// Library/POUs/Additional/MC_ActivateNextCommand/Structures/ActivateNextCommandRecvData
{attribute 'pack_mode' := '1'} 
// ------------------------------------------------------------------------- 
//  SRCI Robot Library                                                
// ------------------------------------------------------------------------- 
//                                                                           
//  Object:      ActivateNextCommandRecvData                                       
//  Author:      Thorsten Brach                                                
//  Date:        2024-06-01
//
//  Description:                                              
//   
//                                                                           
//  Copyright: 
//    (C) 2024 Thorsten Brach. All rights reserved                                                                                                                                            
//             Licensed under the LGPL-3.0 license.
//                                                                           
//  Disclaimer:                                                                           
//    This project is provided without any guarantee and can be used for   
//    private and commercial purposes. Any use is at the user’s 
//    own risk and responsibility.
//
// -------------------------------------------------------------------------
TYPE ActivateNextCommandRecvData EXTENDS RspHeader :
STRUCT
  /// Relates to ListenerID >0
  /// Number of successful trigger -based command invocations
  /// For more information refer to chapter 5.5.12.4.
  InvocationCounter  : USINT;
  /// Reserve
  Reserve            : SINT;
  /// Unique system-generated ID of the "Action" when the function is triggered.
  /// • >0: The "Action" is started by the trigger function with identical FollowID.
  /// • <0: The "Action" is stopped by the trigger function with identical FollowID.
  /// For more information see chapter 5.5.12.4 EmitterID, ListenerID, FollowID and OriginID
  OriginID           : INT;
END_STRUCT
END_TYPE

// Library/POUs/Additional/MC_ActivateNextCommand/Structures/ActivateNextCommandSendData
{attribute 'pack_mode' := '1'}
// ------------------------------------------------------------------------- 
//  SRCI Robot Library                                                
// ------------------------------------------------------------------------- 
//                                                                           
//  Object:      ActivateNextCommandParCmd                                       
//  Author:      Thorsten Brach                                                
//  Date:        2024-06-01
//
//  Description:                                              
//   
//                                                                           
//  Copyright: 
//    (C) 2024 Thorsten Brach. All rights reserved                                                                                                                                            
//             Licensed under the LGPL-3.0 license.
//                                                                           
//  Disclaimer:                                                                           
//    This project is provided without any guarantee and can be used for   
//    private and commercial purposes. Any use is at the user’s 
//    own risk and responsibility.
//
// -------------------------------------------------------------------------
TYPE ActivateNextCommandSendData EXTENDS CmdHeader:   
STRUCT  
  /// ID of Action that will be executed when this command is active
  /// • >0: Start Action        - Start executing the Action function with the identical ListenerID.
  /// • <0: Stop Action         - Stop executing the Action function with the identical ListenerID.
  /// •  0: Undefined (default) - If no EmitterID is defined, the function returns an error message
  /// For more information see chapter 5.5.12.4
  EmitterID  : ARRAY[0..3] OF SINT;  
  /// ID of the trigger function that may be triggered:
  /// • 0: Immediately (default). - Start executing THIS function immediately.
  /// • >0: Triggero Start executing when the trigger function with the identical EmitterID is called.
  /// For more information see chapter 5.5.12.4.
  ListenerID : SINT;
  /// Reserve
  Reserve    : BYTE;
END_STRUCT
END_TYPE

// Library/POUs/Additional/MC_AvoidSingularity/Structures/AvoidSingularityOutCmd
{attribute 'pack_mode' := '1'} 
// ------------------------------------------------------------------------- 
//  SRCI Robot Library                                                
// ------------------------------------------------------------------------- 
//                                                                           
//  Object:      AvoidSingularityOutCmd                                       
//  Author:      Thorsten Brach                                                
//  Date:        2024-06-22
//
//  Description:                                              
//   
//                                                                           
//  Copyright: 
//    (C) 2024 Thorsten Brach. All rights reserved                                                                                                                                            
//             Licensed under the LGPL-3.0 license.
//                                                                           
//  Disclaimer:                                                                           
//    This project is provided without any guarantee and can be used for   
//    private and commercial purposes. Any use is at the user’s 
//    own risk and responsibility.
//
// -------------------------------------------------------------------------
TYPE AvoidSingularityOutCmd :
STRUCT
END_STRUCT
END_TYPE

// Library/POUs/Additional/MC_AvoidSingularity/Structures/AvoidSingularityParCmd
{attribute 'pack_mode' := '1'} 
// ------------------------------------------------------------------------- 
//  SRCI Robot Library                                                
// ------------------------------------------------------------------------- 
//                                                                           
//  Object:      AvoidSingularityParCmd                                       
//  Author:      Thorsten Brach                                                
//  Date:        2024-06-22
//
//  Description:                                              
//   
//                                                                           
//  Copyright: 
//    (C) 2024 Thorsten Brach. All rights reserved                                                                                                                                            
//             Licensed under the LGPL-3.0 license.
//                                                                           
//  Disclaimer:                                                                           
//    This project is provided without any guarantee and can be used for   
//    private and commercial purposes. Any use is at the user’s 
//    own risk and responsibility.
//
// -------------------------------------------------------------------------
TYPE AvoidSingularityParCmd :
STRUCT
  /// Define in which way the singularity should be avoided
  Mode : SingularityAvoidanceMode; 
END_STRUCT
END_TYPE

// Library/POUs/Additional/MC_AvoidSingularity/Structures/AvoidSingularityRecvData
{attribute 'pack_mode' := '1'} 
// ------------------------------------------------------------------------- 
//  SRCI Robot Library                                                
// ------------------------------------------------------------------------- 
//                                                                           
//  Object:      AvoidSingularityRecvData                                       
//  Author:      Thorsten Brach                                                
//  Date:        2024-06-22
//
//  Description:                                              
//   
//                                                                           
//  Copyright: 
//    (C) 2024 Thorsten Brach. All rights reserved                                                                                                                                            
//             Licensed under the LGPL-3.0 license.
//                                                                           
//  Disclaimer:                                                                           
//    This project is provided without any guarantee and can be used for   
//    private and commercial purposes. Any use is at the user’s 
//    own risk and responsibility.
//
// -------------------------------------------------------------------------
TYPE AvoidSingularityRecvData EXTENDS RspHeader :
STRUCT
  /// TRUE when robot is set to RA power state "Enabled".
  Enabled : BOOL;
END_STRUCT
END_TYPE

// Library/POUs/Additional/MC_AvoidSingularity/Structures/AvoidSingularitySendData
{attribute 'pack_mode' := '1'}
// ------------------------------------------------------------------------- 
//  SRCI Robot Library                                                
// ------------------------------------------------------------------------- 
//                                                                           
//  Object:      AvoidSingularitySendData                                       
//  Author:      Thorsten Brach                                                
//  Date:        2024-06-22
//
//  Description:                                              
//   
//                                                                           
//  Copyright: 
//    (C) 2024 Thorsten Brach. All rights reserved                                                                                                                                            
//             Licensed under the LGPL-3.0 license.
//                                                                           
//  Disclaimer:                                                                           
//    This project is provided without any guarantee and can be used for   
//    private and commercial purposes. Any use is at the user’s 
//    own risk and responsibility.
//
// -------------------------------------------------------------------------
TYPE AvoidSingularitySendData EXTENDS CmdHeader: 
STRUCT
  /// Set TRUE to activate avoid singularity mode
  Enable : BOOL;
  /// Define in which way the singularity should be avoided
  Mode   : SingularityAvoidanceMode;
END_STRUCT
END_TYPE

// Library/POUs/Additional/MC_BrakeTest/Structures/BrakeTestOutCmd
{attribute 'pack_mode' := '1'} 
// ------------------------------------------------------------------------- 
//  SRCI Robot Library                                                
// ------------------------------------------------------------------------- 
//                                                                           
//  Object:      BrakeTestOutCmd                                       
//  Author:      Thorsten Brach                                                
//  Date:        2024-06-01
//
//  Description:                                              
//   
//                                                                           
//  Copyright: 
//    (C) 2024 Thorsten Brach. All rights reserved                                                                                                                                            
//             Licensed under the LGPL-3.0 license.
//                                                                           
//  Disclaimer:                                                                           
//    This project is provided without any guarantee and can be used for   
//    private and commercial purposes. Any use is at the user’s 
//    own risk and responsibility.
//
// -------------------------------------------------------------------------
TYPE BrakeTestOutCmd :
STRUCT
  /// Indicates the result of the brake test of the robot axes related to the brake test.
  /// • TRUE: The brake test has been realized successfully.
  /// • FALSE: The brake test failed. 
  /// See Table 6-735 for bit assignment.
  RobotAxesStatus    : RobotAxesFlags;
  /// Indicates the result of the brake test of the external robot axes related to the brake test.
  /// • TRUE: The brake test has been realized successfully.
  /// • FALSE: The brake test failed.
  /// See Table 6-735 for bit assignment.
  ExternalAxesStatus : ExternalAxesFlags;
  /// Indicates the warning messages availability related to the brake functionality of the robot axes reported by the RC.
  /// • TRUE: One or more warning messages are available.
  /// • FALSE: No warning message is available.
  /// See Table 6-735 for bit assignment.
  RobotAxesWarning   : RobotAxesFlags;
  /// Indicates the warning messages availability related to the brake functionality of the external robot axis reported by the RC.
  /// • TRUE: One or more warning messages are available.
  /// • FALSE: No warning message is available.
  /// See Table 6-735 for bit assignment.
  ExternalAxesWarning: ExternalAxesFlags;
END_STRUCT
END_TYPE

// Library/POUs/Additional/MC_BrakeTest/Structures/BrakeTestParCmd
{attribute 'pack_mode' := '1'} 
// ------------------------------------------------------------------------- 
//  SRCI Robot Library                                                
// ------------------------------------------------------------------------- 
//                                                                           
//  Object:      BrakeTestParCmd                                       
//  Author:      Thorsten Brach                                                
//  Date:        2024-06-01
//
//  Description:                                              
//   
//                                                                           
//  Copyright: 
//    (C) 2024 Thorsten Brach. All rights reserved                                                                                                                                            
//             Licensed under the LGPL-3.0 license.
//                                                                           
//  Disclaimer:                                                                           
//    This project is provided without any guarantee and can be used for   
//    private and commercial purposes. Any use is at the user’s 
//    own risk and responsibility.
//
// -------------------------------------------------------------------------
TYPE BrakeTestParCmd :
STRUCT
  /// Parameter which determines the behavior towards the previously sent and still active or buffered commands.
  AbortingMode       : AbortingMode;
  /// Defines which of the robot axis should be activated for the brake test.
  /// • TRUE (default): Axis activated.
  /// • FALSE: Axis deactivated.
  /// See Table 6-735 for bit assignment.
  RobotAxesActive    : RobotAxesFlags;
  /// Defines which of the external robot axis should be activated for the brake test.
  /// • TRUE: Axis activated.
  /// • FALSE (default): Axis deactivated.
  /// See Table 6-735 for bit assignment.   
  ExternalAxesActive : ExternalAxesFlags;
  /// Defines the target sequence in which the command will be executed
  SequenceFlag       : SequenceFlag;
END_STRUCT
END_TYPE

// Library/POUs/Additional/MC_BrakeTest/Structures/BrakeTestRecvData
{attribute 'pack_mode' := '1'} 
// ------------------------------------------------------------------------- 
//  SRCI Robot Library                                                
// ------------------------------------------------------------------------- 
//                                                                           
//  Object:      BrakeTestRecvData                                       
//  Author:      Thorsten Brach                                                
//  Date:        2024-06-01
//
//  Description:                                              
//   
//                                                                           
//  Copyright: 
//    (C) 2024 Thorsten Brach. All rights reserved                                                                                                                                            
//             Licensed under the LGPL-3.0 license.
//                                                                           
//  Disclaimer:                                                                           
//    This project is provided without any guarantee and can be used for   
//    private and commercial purposes. Any use is at the user’s 
//    own risk and responsibility.
//
// -------------------------------------------------------------------------
TYPE BrakeTestRecvData EXTENDS RspHeader :
STRUCT
  /// Indicates the result of the brake test of the robot axes related to the brake test.
  /// • TRUE: The brake test has been realized successfully.
  /// • FALSE: The brake test failed. 
  /// See Table 6-735 for bit assignment.
  RobotAxesStatus    : BYTE;
  /// Indicates the result of the brake test of the external robot axes related to the brake test.
  /// • TRUE: The brake test has been realized successfully.
  /// • FALSE: The brake test failed.
  /// See Table 6-735 for bit assignment.
  ExternalAxesStatus : BYTE;
  /// Indicates the warning messages availability related to the brake functionality of the robot axes reported by the RC.
  /// • TRUE: One or more warning messages are available.
  /// • FALSE: No warning message is available.
  /// See Table 6-735 for bit assignment.
  RobotAxesWarning   : BYTE;
  /// Indicates the warning messages availability related to the brake functionality of the external robot axis reported by the RC.
  /// • TRUE: One or more warning messages are available.
  /// • FALSE: No warning message is available.
  /// See Table 6-735 for bit assignment.
  ExternalAxesWarning: BYTE;
END_STRUCT
END_TYPE

// Library/POUs/Additional/MC_BrakeTest/Structures/BrakeTestSendData
{attribute 'pack_mode' := '1'}
// ------------------------------------------------------------------------- 
//  SRCI Robot Library                                                
// ------------------------------------------------------------------------- 
//                                                                           
//  Object:      BrakeTestSendData                                       
//  Author:      Thorsten Brach                                                
//  Date:        2024-06-01
//
//  Description:                                              
//   
//                                                                           
//  Copyright: 
//    (C) 2024 Thorsten Brach. All rights reserved                                                                                                                                            
//             Licensed under the LGPL-3.0 license.
//                                                                           
//  Disclaimer:                                                                           
//    This project is provided without any guarantee and can be used for   
//    private and commercial purposes. Any use is at the user’s 
//    own risk and responsibility.
//
// -------------------------------------------------------------------------
TYPE BrakeTestSendData EXTENDS CmdHeader:   
STRUCT
  /// Defines which of the robot axis should be activated for the brake test.
  /// • TRUE (default): Axis activated.
  /// • FALSE: Axis deactivated.
  /// See Table 6-735 for bit assignment.
  RobotAxesActive    : BYTE;
  /// Defines which of the external robot axis should be activated for the brake test.
  /// • TRUE: Axis activated.
  /// • FALSE (default): Axis deactivated.
  /// See Table 6-735 for bit assignment.   
  ExternalAxesActive : BYTE; 
END_STRUCT
END_TYPE

// Library/POUs/Additional/MC_CallSubprogram/Structures/CallSubprogramOutCmd
{attribute 'pack_mode' := '1'} 
// ------------------------------------------------------------------------- 
//  SRCI Robot Library                                                
// ------------------------------------------------------------------------- 
//                                                                           
//  Object:      CallSubprogramOutCmd                                       
//  Author:      Thorsten Brach                                                
//  Date:        2024-08-03
//
//  Description:                                              
//   
//                                                                           
//  Copyright: 
//    (C) 2024 Thorsten Brach. All rights reserved                                                                                                                                            
//             Licensed under the LGPL-3.0 license.
//                                                                           
//  Disclaimer:                                                                           
//    This project is provided without any guarantee and can be used for   
//    private and commercial purposes. Any use is at the user’s 
//    own risk and responsibility.
//
// -------------------------------------------------------------------------
TYPE CallSubprogramOutCmd :
STRUCT
  /// Unique, system-generated ID of the instance of CallSubprogram. 
  /// Can be used to specifically stop instance of a subprogram via the function Stop Subprogram (chapter 6.5.21) 
  /// if multiinstancing  is supported by RC 
  InstanceID         : DINT; 
  /// Unique system-generated ID of the "Action" when the function is triggered.
  /// • >0: The "Action" is started by the trigger function with identical FollowID.
  /// • <0: The "Action" is stopped by the trigger function with identical FollowID.
  /// For more information see chapter 5.5.12.4 EmitterID, ListenerID, FollowID and OriginID
  OriginID           : INT;
  /// Relates to ListenerID >0
  /// Number of successful trigger -based command invocations
  /// For more information refer to chapter 5.5.12.4.
  InvocationCounter  : USINT;
  /// The requested subprogram on the RC is in progress. Movement of the axes trough this subprogram is possible.
  InProgress         : BOOL;
  /// Acyclic output parameters of the subprogram Array length adjusts to transmitted data (max 190 bytes)
  ReturnData         : ARRAY[0..RobotLibraryParameter.SUB_PROGRAM_DATA_MAX] OF BYTE;
END_STRUCT
END_TYPE

// Library/POUs/Additional/MC_CallSubprogram/Structures/CallSubprogramParCmd
{attribute 'pack_mode' := '1'} 
// ------------------------------------------------------------------------- 
//  SRCI Robot Library                                                
// ------------------------------------------------------------------------- 
//                                                                           
//  Object:      CallSubprogramParCmd                                       
//  Author:      Thorsten Brach                                                
//  Date:        2024-08-03
//
//  Description:                                              
//   
//                                                                           
//  Copyright: 
//    (C) 2024 Thorsten Brach. All rights reserved                                                                                                                                            
//             Licensed under the LGPL-3.0 license.
//                                                                           
//  Disclaimer:                                                                           
//    This project is provided without any guarantee and can be used for   
//    private and commercial purposes. Any use is at the user’s 
//    own risk and responsibility.
//
// -------------------------------------------------------------------------
TYPE CallSubprogramParCmd :
STRUCT
  /// Program number of the subprogram in the RC
  JobID             : UINT;
  /// ID of associated trigger function:
  /// • 0: No Trigger (default) - No trigger related behavior
  /// • >0: Triggero - Start executing when the trigger function with the identical EmitterID is triggered.
  /// Always positive.
  /// For more information, see chapter 5.5.12 Triggers
  ListenerID        : SINT;
  /// Acyclic input parameters of the subprogram Array length adjusts to transmitted data (max 190 bytes)
  Data              : ARRAY[0..RobotLibraryParameter.SUB_PROGRAM_DATA_MAX] OF BYTE;
END_STRUCT
END_TYPE

// Library/POUs/Additional/MC_CallSubprogram/Structures/CallSubprogramRecvData
{attribute 'pack_mode' := '1'} 
// ------------------------------------------------------------------------- 
//  SRCI Robot Library                                                
// ------------------------------------------------------------------------- 
//                                                                           
//  Object:      CallSubprogramRecvData                                       
//  Author:      Thorsten Brach                                                
//  Date:        2024-08-03
//
//  Description:                                              
//   
//                                                                           
//  Copyright: 
//    (C) 2024 Thorsten Brach. All rights reserved                                                                                                                                            
//             Licensed under the LGPL-3.0 license.
//                                                                           
//  Disclaimer:                                                                           
//    This project is provided without any guarantee and can be used for   
//    private and commercial purposes. Any use is at the user’s 
//    own risk and responsibility.
//
// -------------------------------------------------------------------------
TYPE CallSubprogramRecvData EXTENDS RspHeader :
STRUCT
  /// Relates to ListenerID >0
  /// Number of successful trigger-based command invocations - For more information refer TO chapter 5.5.12.4
  InvocationCounter : USINT;  
  /// Reserve
  Reserve           : SINT;
  /// Unique system-generated ID of the "Action" when the function is triggered.
  /// • >0: The "Action" is started by the trigger funcrion with identical FollowID.
  /// • <0: The "Action" is stopped by the trigger function with identical FollowID.
  /// For more information see chapter 5.5.12.4 EmitterID, ListenerID, FollowID and OriginID
  OriginID          : INT;
  /// Percentage of already traversed distance of current job.
  /// If not supported : • -1
  Progress          : UINT;
  /// The requested subprogram on the RC is in progress. Movement of the axes trough this subprogram is possible.
  InProgress        : BOOL;
  /// Acyclic output parameters of the subprogram Array length adjusts to transmitted data (max 190 bytes)
  ReturnData        : ARRAY[0..RobotLibraryParameter.SUB_PROGRAM_DATA_MAX] OF BYTE;  
END_STRUCT
END_TYPE

// Library/POUs/Additional/MC_CallSubprogram/Structures/CallSubprogramSendData
{attribute 'pack_mode' := '1'}
// ------------------------------------------------------------------------- 
//  SRCI Robot Library                                                
// ------------------------------------------------------------------------- 
//                                                                           
//  Object:      CallSubprogramSendData                                       
//  Author:      Thorsten Brach                                                
//  Date:        2024-08-03
//
//  Description:                                              
//   
//                                                                           
//  Copyright: 
//    (C) 2024 Thorsten Brach. All rights reserved                                                                                                                                            
//             Licensed under the LGPL-3.0 license.
//                                                                           
//  Disclaimer:                                                                           
//    This project is provided without any guarantee and can be used for   
//    private and commercial purposes. Any use is at the user’s 
//    own risk and responsibility.
//
// -------------------------------------------------------------------------
TYPE CallSubprogramSendData EXTENDS CmdHeader: 
STRUCT
  /// ID of Action that will be executed when this command is active
  /// • >0: Start Action - Start executing the Action function with the identical ListenerID.
  /// • <0: Stop Action  -  Stop executing the Action function with the identical ListenerID.
  /// • 0: No trigger (default)-  If no EmitterID is defined, the function will not trigger any Action during its execution
  /// For more information see section Triggers of this chapter or chapter 5.5.12.4.
  EmitterID          : ARRAY [0..3] OF SINT;  
  /// ID of associated trigger function:
  /// • 0: No Trigger (default) - No trigger related behavior
  /// • >0: Triggero - Start executing when the trigger function with the identical EmitterID is triggered.
  /// Always positive.
  /// For more information, see chapter 5.5.12 Triggers
  ListenerID        : SINT;
  /// Reserve
  Reserve           : BYTE;
  /// Program number of the subprogram in the RC
  JobID             : UINT;
  /// Acyclic input parameters of the subprogram Array length adjusts to transmitted data (max 190 bytes)
  Data              : ARRAY[0..RobotLibraryParameter.SUB_PROGRAM_DATA_MAX] OF BYTE;
END_STRUCT
END_TYPE

// Library/POUs/Additional/MC_CollisionDetection/Structures/CollisionDetectionOutCmd
{attribute 'pack_mode' := '1'} 
// ------------------------------------------------------------------------- 
//  SRCI Robot Library                                                
// ------------------------------------------------------------------------- 
//                                                                           
//  Object:      CollisionDetectionOutCmd                                       
//  Author:      Thorsten Brach                                                
//  Date:        2024-06-22
//
//  Description:                                              
//   
//                                                                           
//  Copyright: 
//    (C) 2024 Thorsten Brach. All rights reserved                                                                                                                                            
//             Licensed under the LGPL-3.0 license.
//                                                                           
//  Disclaimer:                                                                           
//    This project is provided without any guarantee and can be used for   
//    private and commercial purposes. Any use is at the user’s 
//    own risk and responsibility.
//
// -------------------------------------------------------------------------
TYPE CollisionDetectionOutCmd :
STRUCT
END_STRUCT
END_TYPE

// Library/POUs/Additional/MC_CollisionDetection/Structures/CollisionDetectionParCmd
{attribute 'pack_mode' := '1'} 
// ------------------------------------------------------------------------- 
//  SRCI Robot Library                                                
// ------------------------------------------------------------------------- 
//                                                                           
//  Object:      CollisionDetectionParCmd                                       
//  Author:      Thorsten Brach                                                
//  Date:        2024-06-22
//
//  Description:                                              
//   
//                                                                           
//  Copyright: 
//    (C) 2024 Thorsten Brach. All rights reserved                                                                                                                                            
//             Licensed under the LGPL-3.0 license.
//                                                                           
//  Disclaimer:                                                                           
//    This project is provided without any guarantee and can be used for   
//    private and commercial purposes. Any use is at the user’s 
//    own risk and responsibility.
//
// -------------------------------------------------------------------------
TYPE CollisionDetectionParCmd :
STRUCT
  /// Processing mode
  ProcessingMode     : ProcessingMode;
  ///  Defines the robot behavior after detecting the collision (at least one option must be supported):
  ReactionMode       : CollisionReactionMode;
  /// Set TRUE to activate and FALSE to deactivate "CollisionDetection".
  /// Default: TRUE
  ActivateMonitoring : BOOL;
  /// Defines the type of threshold setting (at least one option must be supported)
  ThresholdMode      : ThresholdMode;
  /// Defines the level of sensitivity of all axes.
  /// • 0..99: Sensitivity lower than robot vendor default. 
  ///          At minimum value "0" there is no sensitivity. The lower the value, the lower the sensitivity at the collision detection.
  /// • 100 (default): The value is aligned with the robot vendor-specific default value.
  /// • 101..200: Sensitivity higher than robot vendor default. At maximum value "200" highest possible sensitivity at the collision detection.
  Sensitivity        : REAL;
  /// Defines the level of sensitivity of the respective axis.
  /// Values:
  /// • 0..99: Sensitivity lower than robot vendor default. At minimum value "0" there is no sensitivity and collision detection for the respective axis. 
  ///          The lower the value, the lower the sensitivity at the collision detection.
  /// • 100 (default): The value is aligned with the robot vendor-specific default value.
  /// • 101..200: Sensitivity higher than robot vendor default. At maximum value "200" highest possible sensitivity at the collision detection.
  /// Index:
  /// • [0]: J1 First joint of the robot.
  /// • [1]: J2 Second joint of the robot.
  /// • [2] J3 Third joint of the robot.
  /// • [3] J4 Forth joint of the robot.
  /// • [4] J5 Fifth joint of the robot.
  /// • [5] J6 Six joint of the robot.
  /// • [6] J7 Seventh joint of the robot, if willbe used.
  SensitivityAxis    : ARRAY[0..6] OF REAL;
  /// Relates to "ThresholdMode" Manual. Defines the threshold of the torque for each robot axis. If the threshold is exceeded, the RA stops.
  /// Index:
  /// • [0] J1 First joint of the robot.
  /// • [1] J2 Second joint of the robot.
  /// • [2] J3 Third joint of the robot.
  /// • [3] J4 Forth joint of the robot.
  /// • [4] J5 Fifth joint of the robot.
  /// • [5] J6 Six joint of the robot.
  /// • [6] J7 Seventh joint of the robot, if will be used
  LimitAxis          : ARRAY[0..6] OF REAL;
  /// Relates to "LimitAxis". Defines the unit of the threshold.
  /// • [0]: Percentage (%) (default) O
  /// • [1]: Newton meter (Nm). O
  /// • [2] Milliampere (mA).
  UnitLimitAxis      : USINT;
  /// Defines the target sequence in which the command will be executed
  SequenceFlag       : SequenceFlag;
END_STRUCT
END_TYPE

// Library/POUs/Additional/MC_CollisionDetection/Structures/CollisionDetectionRecvData
{attribute 'pack_mode' := '1'} 
// ------------------------------------------------------------------------- 
//  SRCI Robot Library                                                
// ------------------------------------------------------------------------- 
//                                                                           
//  Object:      CollisionDetectionRecvData                                       
//  Author:      Thorsten Brach                                                
//  Date:        2024-06-22
//
//  Description:                                              
//   
//                                                                           
//  Copyright: 
//    (C) 2024 Thorsten Brach. All rights reserved                                                                                                                                            
//             Licensed under the LGPL-3.0 license.
//                                                                           
//  Disclaimer:                                                                           
//    This project is provided without any guarantee and can be used for   
//    private and commercial purposes. Any use is at the user’s 
//    own risk and responsibility.
//
// -------------------------------------------------------------------------
TYPE CollisionDetectionRecvData EXTENDS RspHeader :
STRUCT
END_STRUCT
END_TYPE

// Library/POUs/Additional/MC_CollisionDetection/Structures/CollisionDetectionSendData
{attribute 'pack_mode' := '1'}
// ------------------------------------------------------------------------- 
//  SRCI Robot Library                                                
// ------------------------------------------------------------------------- 
//                                                                           
//  Object:      CollisionDetectionSendData                                       
//  Author:      Thorsten Brach                                                
//  Date:        2024-06-22
//
//  Description:                                              
//   
//                                                                           
//  Copyright: 
//    (C) 2024 Thorsten Brach. All rights reserved                                                                                                                                            
//             Licensed under the LGPL-3.0 license.
//                                                                           
//  Disclaimer:                                                                           
//    This project is provided without any guarantee and can be used for   
//    private and commercial purposes. Any use is at the user’s 
//    own risk and responsibility.
//
// -------------------------------------------------------------------------
TYPE CollisionDetectionSendData EXTENDS CmdHeader: 
STRUCT
  /// Set TRUE to activate and FALSE to deactivate "CollisionDetection".
  /// Default: TRUE
  ActivateMonitoring : BOOL;
  /// Relates to "LimitAxis". Defines the unit of the threshold.
  /// • [0]: Percentage (%) (default) O
  /// • [1]: Newton meter (Nm). O
  /// • [2] Milliampere (mA).
  UnitLimitAxis      : USINT;
  /// Defines the type of threshold setting (at least one option must be supported)
  ThresholdMode      : ThresholdMode;
  ///  Defines the robot behavior after detecting the collision (at least one option must be supported):
  ReactionMode       : CollisionReactionMode;
  /// Defines the level of sensitivity of all axes.
  /// • 0..99: Sensitivity lower than robot vendor default. 
  ///          At minimum value "0" there is no sensitivity. The lower the value, the lower the sensitivity at the collision detection.
  /// • 100 (default): The value is aligned with the robot vendor-specific default value.
  /// • 101..200: Sensitivity higher than robot vendor default. At maximum value "200" highest possible sensitivity at the collision detection.
  Sensitivity        : INT;
  /// Defines the level of sensitivity of the respective axis.
  /// Values:
  /// • 0..99: Sensitivity lower than robot vendor default. At minimum value "0" there is no sensitivity and collision detection for the respective axis. 
  ///          The lower the value, the lower the sensitivity at the collision detection.
  /// • 100 (default): The value is aligned with the robot vendor-specific default value.
  /// • 101..200: Sensitivity higher than robot vendor default. At maximum value "200" highest possible sensitivity at the collision detection.
  /// Index:
  /// • [0]: J1 First joint of the robot.
  /// • [1]: J2 Second joint of the robot.
  /// • [2] J3 Third joint of the robot.
  /// • [3] J4 Forth joint of the robot.
  /// • [4] J5 Fifth joint of the robot.
  /// • [5] J6 Six joint of the robot.
  /// • [6] J7 Seventh joint of the robot, if willbe used.
  SensitivityAxis    : ARRAY[0..6] OF INT;

  /// Relates to "ThresholdMode" Manual. Defines the threshold of the torque for each robot axis. If the threshold is exceeded, the RA stops.
  /// Index:
  /// • [0] J1 First joint of the robot.
  /// • [1] J2 Second joint of the robot.
  /// • [2] J3 Third joint of the robot.
  /// • [3] J4 Forth joint of the robot.
  /// • [4] J5 Fifth joint of the robot.
  /// • [5] J6 Six joint of the robot.
  /// • [6] J7 Seventh joint of the robot, if will be used
  LimitAxis          : ARRAY[0..6] OF REAL;
END_STRUCT
END_TYPE

// Library/POUs/Additional/MC_ExchangeConfiguration/Structures/ExchangeConfigurationOutCmd
{attribute 'pack_mode' := '1'} 
// ------------------------------------------------------------------------- 
//  SRCI Robot Library                                                
// ------------------------------------------------------------------------- 
//                                                                           
//  Object:      ExchangeConfigurationOutCmd                                       
//  Author:      Thorsten Brach                                                
//  Date:        2024-06-22
//
//  Description:                                              
//   
//                                                                           
//  Copyright: 
//    (C) 2024 Thorsten Brach. All rights reserved                                                                                                                                            
//             Licensed under the LGPL-3.0 license.
//                                                                           
//  Disclaimer:                                                                           
//    This project is provided without any guarantee and can be used for   
//    private and commercial purposes. Any use is at the user’s 
//    own risk and responsibility.
//
// -------------------------------------------------------------------------
TYPE ExchangeConfigurationOutCmd :
STRUCT
  /// Returns a metric of how many CMDs it can receive and manage at the same time
  LengthACR                 : UINT;
  /// Highest index of available tools on the RC.
  HighestToolIndex          : USINT;
  /// Highest index of available frames on the RC.
  HighestFrameIndex         : USINT;
  /// Highest index of available loads on the RC.
  HighestLoadIndex          : USINT;
  /// Highest index of available work areas on the RC.
  HighestWorkAreaIndex      : USINT;
  /// Datas which are synchronized
  DataInSync                : DataInSync;
  /// Index of tool changed on RC
  ChangeIndexTool           : USINT;
  /// Index of frame changed on RC
  ChangeIndexFrame          : USINT;
  /// Index of load changed on RC
  ChangeIndexLoad           : USINT;
  ///Index of work area changed on RC
  ChangeIndexWorkArea       : USINT;
  /// Working hours of an RA connected to the RC
  RAWorkingHours            : UDINT;
  /// Signals that a brake test is required in the defined monitoring time (see chapter 6.5.27)
  BrakeTestRequired         : BOOL;
  /// StepMode is active and set to ExactStop (see chapter 6.1.3)
  StepModeExactStopActive   : BOOL;
  /// StepMode is active and set to Blending (see chapter 6.1.3)
  StepModeBlendingActive    : BOOL;
  /// PathAccuracyMode is active (see chapter 6.5.22)
  PathAccuracyMode          : BOOL;
  /// AvoidSingularity is active (see chapter 6.5.23)
  AvoidSingularity          : BOOL;
  /// CollisionDetection is active (see chapter 6.5.35)
  CollisionDetectionEnabled : BOOL;
  /// Cyclic dynamics status bit Accelerating is supported by RC (see chapter 5.5.3.2)
  AcceleratingSupported     : BOOL;
  /// Cyclic dynamics status bit Decelerating is supported by RC (see chapter 5.5.3.2)
  DecceleratingSupported    : BOOL;
  /// Cyclic dynamics status bit ConstantVelocity is supported by RC (see chapter 5.5.3.2)
  ConstantVelocitySupported : BOOL;
  /// Total system hours of an RA connected to the RC. Must not be modifiable by the user.
  /// •  0: Invalid
  /// • >1: Total system hours
  RCWorkingHours            : UDINT;
END_STRUCT
END_TYPE

// Library/POUs/Additional/MC_ExchangeConfiguration/Structures/ExchangeConfigurationParCmd
{attribute 'pack_mode' := '1'} 
// ------------------------------------------------------------------------- 
//  SRCI Robot Library                                                
// ------------------------------------------------------------------------- 
//                                                                           
//  Object:      ExchangeConfigurationParCmd                                       
//  Author:      Thorsten Brach                                                
//  Date:        2024-06-22
//
//  Description:                                              
//   
//                                                                           
//  Copyright: 
//    (C) 2024 Thorsten Brach. All rights reserved                                                                                                                                            
//             Licensed under the LGPL-3.0 license.
//                                                                           
//  Disclaimer:                                                                           
//    This project is provided without any guarantee and can be used for   
//    private and commercial purposes. Any use is at the user’s 
//    own risk and responsibility.
//
// -------------------------------------------------------------------------
TYPE ExchangeConfigurationParCmd :
STRUCT
  /// Defines up to which level of severity messages will be logged in the RC's server log
  LogLevel                   : LogLevel;
  /// Defines blending behavior for single move commands. One of the optional modes must be supported.
  ///  • 0 (default): Move to end position
  ///       Robot moves exactly the target position independently of the selected "BlendingMode"
  ///  • 1: Wait at blending parameter 
  ///       Robot stops its movement when the specified blending parameter is reached
  WaitAtBlendingZone         : BOOL;
  /// Allow a sequence switch from primary to secondary while a subprogram called via CallSubprogram (6.5.18) in the sequence is in progress
  AllowSecSeqWhileSubprogram : BOOL;
  /// Allows blending when CallSubprogram is called in sequence and removed afterwards. For more information see chapter 6.5.21.
  /// • 0 (default): Dynamic blending is prevented
  /// • 1: Dynamic blending is allowed
  AllowDynamicBlending       : BOOL;
  /// Defines waiting time of RC between receiving a first move command when motion queue is empty and starting the first movement. See also chapter 5.6.8.
  DelayTime                  : UINT;
  /// Define number of points required to calculate the blending. See also chapter 5.6.8.
  WaitForNrOfCmd             : UINT;
  /// Maximum allowed time between incrementation of LifeSign before communication error.
  /// • <10 ms: Invalid
  /// • 50 ms: default
  /// See also chapter 5.6.6.2.
  LifeSignTimeOut            : UINT;
  /// Defines a delay time between detecting an inconsistency of configuration data between server and client and executing the defined SyncReaction. 
  /// Always positive. Default: 0 ms
  SyncDelay                  : UINT;
  /// Specifies system reaction in case inconsistency of synchronization data is detected according to Table 6-81. For more information refer to chapter 5.6.7.2
  SyncReaction               : SyncReaction;
  /// Datas which are synchronized
  DataInSync                 : DataInSync;
  /// Enable datas to synchronize
  DataEnableSync             : DataEnableSync;
END_STRUCT
END_TYPE

// Library/POUs/Additional/MC_ExchangeConfiguration/Structures/ExchangeConfigurationRecvData
{attribute 'pack_mode' := '1'} 
// ------------------------------------------------------------------------- 
//  SRCI Robot Library                                                
// ------------------------------------------------------------------------- 
//                                                                           
//  Object:      ExchangeConfigurationRecvData                                       
//  Author:      Thorsten Brach                                                
//  Date:        2024-06-22
//
//  Description:                                              
//   
//                                                                           
//  Copyright: 
//    (C) 2024 Thorsten Brach. All rights reserved                                                                                                                                            
//             Licensed under the LGPL-3.0 license.
//                                                                           
//  Disclaimer:                                                                           
//    This project is provided without any guarantee and can be used for   
//    private and commercial purposes. Any use is at the user’s 
//    own risk and responsibility.
//
// -------------------------------------------------------------------------
TYPE ExchangeConfigurationRecvData EXTENDS RspHeader :
STRUCT
  /// TRUE when function is exchanging data
  Enabled                   : BOOL;
  /// Reserve 
  Reserve1                  : BYTE;
   /// Returns a metric of how many CMDs it can receive and manage at the same time
  LengthACR                 : UINT;
  /// Highest index of available tools on the RC.
  HighestToolIndex          : USINT;
  /// Highest index of available frames on the RC.
  HighestFrameIndex         : USINT;
  /// Highest index of available loads on the RC.
  HighestLoadIndex          : USINT;
  /// Highest index of available work areas on the RC.
  HighestWorkAreaIndex      : USINT; 
  /// Datas which are synchronized
  DataInSync                : DataInSync;
  /// Reserve 
  Reserve2                  : BYTE;
  /// Index of tool changed on RC
  ChangeIndexTool           : USINT;
  /// Index of frame changed on RC
  ChangeIndexFrame          : USINT;
  /// Index of load changed on RC
  ChangeIndexLoad           : USINT;
  ///Index of work area changed on RC
  ChangeIndexWorkArea       : USINT;
  /// Working hours of an RA connected to the RC
  RAWorkingHours            : UDINT;
  /// Status byte
  StatusByte                : BYTE;
  /// Cyclic dynamics status bit ConstantVelocity is supported by RC (see chapter 5.5.3.2)
  ConstantVelocitySupported : BOOL;
  /// Total system hours of an RA connected to the RC. Must not be modifiable by the user.
  /// •  0: Invalid
  /// • >1: Total system hours
  RCWorkingHours            : UDINT;
END_STRUCT
END_TYPE

// Library/POUs/Additional/MC_ExchangeConfiguration/Structures/ExchangeConfigurationSendData
{attribute 'pack_mode' := '1'}
// ------------------------------------------------------------------------- 
//  SRCI Robot Library                                                
// ------------------------------------------------------------------------- 
//                                                                           
//  Object:      ExchangeConfigurationSendData                                       
//  Author:      Thorsten Brach                                                
//  Date:        2024-06-22
//
//  Description:                                              
//   
//                                                                           
//  Copyright: 
//    (C) 2024 Thorsten Brach. All rights reserved                                                                                                                                            
//             Licensed under the LGPL-3.0 license.
//                                                                           
//  Disclaimer:                                                                           
//    This project is provided without any guarantee and can be used for   
//    private and commercial purposes. Any use is at the user’s 
//    own risk and responsibility.
//
// -------------------------------------------------------------------------
TYPE ExchangeConfigurationSendData EXTENDS CmdHeader: 
STRUCT
  /// Defines up to which level of severity messages will be logged in the RC's server log
  LogLevel                   : LogLevel;
  /// Miscellaneous control bits 
  CtrlByte                   : BYTE;
  /// Defines waiting time of RC between receiving a first move command when motion queue is empty and starting the first movement. See also chapter 5.6.8.
  DelayTime                  : UINT;
  /// Define number of points required to calculate the blending. See also chapter 5.6.8.
  WaitForNrOfCmd             : UINT;
  /// Maximum allowed time between incrementation of LifeSign before communication error.
  /// • <10 ms: Invalid
  /// • 50 ms: default
  /// See also chapter 5.6.6.2.
  LifeSignTimeOut            : UINT;
  /// Defines a delay time between detecting an inconsistency of configuration data between server and client and executing the defined SyncReaction. 
  /// Always positive. Default: 0 ms
  SyncDelay                  : UINT;
  /// Specifies system reaction in case inconsistency of synchronization data is detected according to Table 6-81. For more information refer to chapter 5.6.7.2
  SyncReaction               : SyncReaction;
  /// Datas which are synchronized
  DataInSync                 : DataInSync;
  /// Reserve
  Reserve1                   : BYTE;
  /// Enable datas to synchronize
  DataEnableSync             : DataEnableSync;  
  /// Reserve
  Reserve2                   : BYTE;
END_STRUCT
END_TYPE

// Library/POUs/Additional/MC_FreeDrive/Structures/FreeDriveOutCmd
{attribute 'pack_mode' := '1'} 
// ------------------------------------------------------------------------- 
//  SRCI Robot Library                                                
// ------------------------------------------------------------------------- 
//                                                                           
//  Object:      FreeDriveOutCmd                                       
//  Author:      Thorsten Brach                                                
//  Date:        2024-06-22
//
//  Description:                                              
//   
//                                                                           
//  Copyright: 
//    (C) 2024 Thorsten Brach. All rights reserved                                                                                                                                            
//             Licensed under the LGPL-3.0 license.
//                                                                           
//  Disclaimer:                                                                           
//    This project is provided without any guarantee and can be used for   
//    private and commercial purposes. Any use is at the user’s 
//    own risk and responsibility.
//
// -------------------------------------------------------------------------
TYPE FreeDriveOutCmd :
STRUCT
  /// TRUE when function is exchanging data
  Enabled                   : BOOL;
  /// Returns a metric of how many CMDs it can receive and manage at the same time
  LengthACR                 : UINT;
  /// Highest index of available tools on the RC.
  HighestToolIndex          : USINT;
  /// Highest index of available frames on the RC.
  HighestFrameIndex         : USINT;
  /// Highest index of available loads on the RC.
  HighestLoadIndex          : USINT;
  /// Highest index of available work areas on the RC.
  HighestWorkAreaIndex      : USINT;
  /// Datas which are synchronized
  DataInSync                : DataInSync;
  /// Index of tool changed on RC
  ChangeIndexTool           : USINT;
  /// Index of frame changed on RC
  ChangeIndexFrame          : USINT;
  /// Index of load changed on RC
  ChangeIndexLoad           : USINT;
  ///Index of work area changed on RC
  ChangeIndexWorkArea       : USINT;
  /// Working hours of an RA connected to the RC
  RAWorkingHours            : UDINT;
  /// Signals that a brake test is required in the defined monitoring time (see chapter 6.5.27)
  BrakeTestRequired         : BOOL;
  /// StepMode is active and set to ExactStop (see chapter 6.1.3)
  StepModeExactStopActive   : BOOL;
  /// StepMode is active and set to Blending (see chapter 6.1.3)
  StepModeBlendingActive    : BOOL;
  /// PathAccuracyMode is active (see chapter 6.5.22)
  PathAccuracyMode          : BOOL;
  /// AvoidSingularity is active (see chapter 6.5.23)
  AvoidSingularity          : BOOL;
  /// CollisionDetection is active (see chapter 6.5.35)
  CollisionDetectionEnabled : BOOL;
  /// Cyclic dynamics status bit Accelerating is supported by RC (see chapter 5.5.3.2)
  AcceleratingSupported     : BOOL;
  /// Cyclic dynamics status bit Decelerating is supported by RC (see chapter 5.5.3.2)
  DecceleratingSupported    : BOOL;
  /// Cyclic dynamics status bit ConstantVelocity is supported by RC (see chapter 5.5.3.2)
  ConstantVelocitySupported : BOOL;
  /// Total system hours of an RA connected to the RC. Must not be modifiable by the user.
  /// •  0: Invalid
  /// • >1: Total system hours
  RCWorkingHours            : UDINT;
END_STRUCT
END_TYPE

// Library/POUs/Additional/MC_FreeDrive/Structures/FreeDriveParCmd
{attribute 'pack_mode' := '1'} 
// ------------------------------------------------------------------------- 
//  SRCI Robot Library                                                
// ------------------------------------------------------------------------- 
//                                                                           
//  Object:      FreeDriveParCmd                                       
//  Author:      Thorsten Brach                                                
//  Date:        2024-06-22
//
//  Description:                                              
//   
//                                                                           
//  Copyright: 
//    (C) 2024 Thorsten Brach. All rights reserved                                                                                                                                            
//             Licensed under the LGPL-3.0 license.
//                                                                           
//  Disclaimer:                                                                           
//    This project is provided without any guarantee and can be used for   
//    private and commercial purposes. Any use is at the user’s 
//    own risk and responsibility.
//
// -------------------------------------------------------------------------
TYPE FreeDriveParCmd :
STRUCT
  /// Defines up to which level of severity messages will be logged in the RC's server log
  LogLevel                   : LogLevel;
  /// Defines blending behavior for single move commands. One of the optional modes must be supported.
  ///  • 0 (default): Move to end position
  ///       Robot moves exactly the target position independently of the selected "BlendingMode"
  ///  • 1: Wait at blending parameter 
  ///       Robot stops its movement when the specified blending parameter is reached
  WaitAtBlendingZone         : BOOL;
  /// Allow a sequence switch from primary to secondary while a subprogram called via CallSubprogram (6.5.18) in the sequence is in progress
  AllowSecSeqWhileSubprogram : BOOL;
  /// ToDo
  AllowDynamicBlending       : BOOL;
  /// Defines waiting time of RC between receiving a first move command when motion queue is empty and starting the first movement. See also chapter 5.6.8.
  DelayTime                  : UINT;
  /// Define number of points required to calculate the blending. See also chapter 5.6.8.
  WaitForNrOfCmd             : UINT;
  /// Maximum allowed time between incrementation of LifeSign before communication error.
  /// • <10 ms: Invalid
  /// • 50 ms: default
  /// See also chapter 5.6.6.2.
  LifeSignTimeOut            : UINT;
  /// Defines a delay time between detecting an inconsistency of configuration data between server and client and executing the defined SyncReaction. 
  /// Always positive. Default: 0 ms
  SyncDelay                  : UINT;
  /// Specifies system reaction in case inconsistency of synchronization data is detected according to Table 6-81. For more information refer to chapter 5.6.7.2
  SyncReaction               : SyncReaction;
  /// Datas which are synchronized
  DataInSync                 : DataInSync;
  /// Enable datas to synchronize
  DataEnableSync             : DataEnableSync;
END_STRUCT
END_TYPE

// Library/POUs/Additional/MC_FreeDrive/Structures/FreeDriveRecvData
{attribute 'pack_mode' := '1'} 
// ------------------------------------------------------------------------- 
//  SRCI Robot Library                                                
// ------------------------------------------------------------------------- 
//                                                                           
//  Object:      FreeDriveRecvData                                       
//  Author:      Thorsten Brach                                                
//  Date:        2024-06-22
//
//  Description:                                              
//   
//                                                                           
//  Copyright: 
//    (C) 2024 Thorsten Brach. All rights reserved                                                                                                                                            
//             Licensed under the LGPL-3.0 license.
//                                                                           
//  Disclaimer:                                                                           
//    This project is provided without any guarantee and can be used for   
//    private and commercial purposes. Any use is at the user’s 
//    own risk and responsibility.
//
// -------------------------------------------------------------------------
TYPE FreeDriveRecvData EXTENDS RspHeader :
STRUCT
  /// TRUE when function is exchanging data
  Enabled                   : BOOL;
END_STRUCT
END_TYPE

// Library/POUs/Additional/MC_FreeDrive/Structures/FreeDriveSendData
{attribute 'pack_mode' := '1'}
// ------------------------------------------------------------------------- 
//  SRCI Robot Library                                                
// ------------------------------------------------------------------------- 
//                                                                           
//  Object:      FreeDriveSendData                                       
//  Author:      Thorsten Brach                                                
//  Date:        2024-06-22
//
//  Description:                                              
//   
//                                                                           
//  Copyright: 
//    (C) 2024 Thorsten Brach. All rights reserved                                                                                                                                            
//             Licensed under the LGPL-3.0 license.
//                                                                           
//  Disclaimer:                                                                           
//    This project is provided without any guarantee and can be used for   
//    private and commercial purposes. Any use is at the user’s 
//    own risk and responsibility.
//
// -------------------------------------------------------------------------
TYPE FreeDriveSendData EXTENDS CmdHeader: 
STRUCT
  /// Set TRUE to activate "FreeDrive".
  Enable            : BOOL;
END_STRUCT
END_TYPE

// Library/POUs/Additional/MC_MeasuringInput/Structures/MeasuringInputOutCmd
{attribute 'pack_mode' := '1'} 
// ------------------------------------------------------------------------- 
//  SRCI Robot Library                                                
// ------------------------------------------------------------------------- 
//                                                                           
//  Object:      MeasuringInputOutCmd                                       
//  Author:      Thorsten Brach                                                
//  Date:        2024-06-21
//
//  Description:                                              
//   
//                                                                           
//  Copyright: 
//    (C) 2024 Thorsten Brach. All rights reserved                                                                                                                                            
//             Licensed under the LGPL-3.0 license.
//                                                                           
//  Disclaimer:                                                                           
//    This project is provided without any guarantee and can be used for   
//    private and commercial purposes. Any use is at the user’s 
//    own risk and responsibility.
//
// -------------------------------------------------------------------------
TYPE MeasuringInputOutCmd :
STRUCT
  /// FB is returning a unique ID for the called measurement.
  MeasuringID        : UINT;
  /// Measured robot position value at the rising edge of the digital input in selected coordinate systems (see input parameters ToolNo and FrameNo).
  Measurings         : ARRAY[1..2] OF MeasuringInputResult;  
END_STRUCT
END_TYPE

// Library/POUs/Additional/MC_MeasuringInput/Structures/MeasuringInputParCmd
{attribute 'pack_mode' := '1'} 
// ------------------------------------------------------------------------- 
//  SRCI Robot Library                                                
// ------------------------------------------------------------------------- 
//                                                                           
//  Object:      MeasuringInputParCmd                                       
//  Author:      Thorsten Brach                                                
//  Date:        2024-06-21
//
//  Description:                                              
//   
//                                                                           
//  Copyright: 
//    (C) 2024 Thorsten Brach. All rights reserved                                                                                                                                            
//             Licensed under the LGPL-3.0 license.
//                                                                           
//  Disclaimer:                                                                           
//    This project is provided without any guarantee and can be used for   
//    private and commercial purposes. Any use is at the user’s 
//    own risk and responsibility.
//
// -------------------------------------------------------------------------
TYPE MeasuringInputParCmd :
STRUCT
  /// Type of measurement (at least one option must be supported):
  MeasuringMode      : MeasuringIoMode;
  /// Specifies the desired digital input register. 
  /// More information about the different periphery register can be found in chapter 6.4
  Index              : USINT;
  ///Specifies the desired bit in the digital input register, that should be read. 
  /// More information about the different periphery register can be found in chapter 6.4.
  BitNumber          : USINT;
END_STRUCT
END_TYPE

// Library/POUs/Additional/MC_MeasuringInput/Structures/MeasuringInputRecvData
{attribute 'pack_mode' := '1'} 
// ------------------------------------------------------------------------- 
//  SRCI Robot Library                                                
// ------------------------------------------------------------------------- 
//                                                                           
//  Object:      MeasuringInputRecvData                                       
//  Author:      Thorsten Brach                                                
//  Date:        2024-06-21
//
//  Description:                                              
//   
//                                                                           
//  Copyright: 
//    (C) 2024 Thorsten Brach. All rights reserved                                                                                                                                            
//             Licensed under the LGPL-3.0 license.
//                                                                           
//  Disclaimer:                                                                           
//    This project is provided without any guarantee and can be used for   
//    private and commercial purposes. Any use is at the user’s 
//    own risk and responsibility.
//
// -------------------------------------------------------------------------
TYPE MeasuringInputRecvData EXTENDS RspHeader :
STRUCT
  /// FB is returning a unique ID for the called measurement.
  MeasuringID        : UINT;
  /// Measured robot position value at the rising edge of the digital input in selected coordinate systems (see input parameters ToolNo and FrameNo).
  Measurings         : ARRAY[1..2] OF MeasuringInputResult;  
END_STRUCT
END_TYPE

// Library/POUs/Additional/MC_MeasuringInput/Structures/MeasuringInputSendData
{attribute 'pack_mode' := '1'}
// ------------------------------------------------------------------------- 
//  SRCI Robot Library                                                
// ------------------------------------------------------------------------- 
//                                                                           
//  Object:      MeasuringInputSendData                                       
//  Author:      Thorsten Brach                                                
//  Date:        2024-06-21
//
//  Description:                                              
//   
//                                                                           
//  Copyright: 
//    (C) 2024 Thorsten Brach. All rights reserved                                                                                                                                            
//             Licensed under the LGPL-3.0 license.
//                                                                           
//  Disclaimer:                                                                           
//    This project is provided without any guarantee and can be used for   
//    private and commercial purposes. Any use is at the user’s 
//    own risk and responsibility.
//
// -------------------------------------------------------------------------
TYPE MeasuringInputSendData EXTENDS CmdHeader:   
STRUCT
  /// Type of measurement (at least one option must be supported):
  MeasuringMode      : MeasuringIoMode;
  /// Specifies the desired digital input register. 
  /// More information about the different periphery register can be found in chapter 6.4
  Index              : USINT;
  ///Specifies the desired bit in the digital input register, that should be read. 
  /// More information about the different periphery register can be found in chapter 6.4.
  BitNumber          : USINT;
END_STRUCT
END_TYPE

// Library/POUs/Additional/MC_OpenBrake/Structures/OpenBrakeOutCmd
{attribute 'pack_mode' := '1'} 
// ------------------------------------------------------------------------- 
//  SRCI Robot Library                                                
// ------------------------------------------------------------------------- 
//                                                                           
//  Object:      BrakeTestOutCmd                                       
//  Author:      Thorsten Brach                                                
//  Date:        2024-06-01
//
//  Description:                                              
//   
//                                                                           
//  Copyright: 
//    (C) 2024 Thorsten Brach. All rights reserved                                                                                                                                            
//             Licensed under the LGPL-3.0 license.
//                                                                           
//  Disclaimer:                                                                           
//    This project is provided without any guarantee and can be used for   
//    private and commercial purposes. Any use is at the user’s 
//    own risk and responsibility.
//
// -------------------------------------------------------------------------
TYPE OpenBrakeOutCmd :
STRUCT
  /// TRUE when "OpenBrake" is active.
  Enabled                   : BOOL;  
  /// Indicates the brake release status of the main robot axes.
  /// • TRUE: The brake of the axis is opened.
  /// • FALSE: The brake of the axis is closed.
  /// See Table 6-735 for bit assignment
  RobotAxesBrakeReleased    : RobotAxesFlags;
  /// Indicates the brake release status of the external robot axes.
  /// • TRUE: The brake of the axis is opened.
  /// • FALSE: The brake of the axis is closed/not supported
  /// See Table 6-735 for bit assignment
  ExternalAxesBrakeReleased : ExternalAxesFlags;
END_STRUCT
END_TYPE

// Library/POUs/Additional/MC_OpenBrake/Structures/OpenBrakeParCmd
{attribute 'pack_mode' := '1'} 
// ------------------------------------------------------------------------- 
//  SRCI Robot Library                                                
// ------------------------------------------------------------------------- 
//                                                                           
//  Object:      OpenBrakeParCmd                                       
//  Author:      Thorsten Brach                                                
//  Date:        2024-06-01
//
//  Description:                                              
//   
//                                                                           
//  Copyright: 
//    (C) 2024 Thorsten Brach. All rights reserved                                                                                                                                            
//             Licensed under the LGPL-3.0 license.
//                                                                           
//  Disclaimer:                                                                           
//    This project is provided without any guarantee and can be used for   
//    private and commercial purposes. Any use is at the user’s 
//    own risk and responsibility.
//
// -------------------------------------------------------------------------
TYPE OpenBrakeParCmd :
STRUCT
  /// Defines which brake of the robot axes must be released.
  /// • TRUE: Open the brake of the axis.
  /// • FALSE (default): Close the brake of the axis.
  RobotAxesBrakeRelease    : RobotAxesFlags;
  /// Defines which brake of the external robot axis must be released.
  /// • TRUE: Open the brake of the axis.
  /// • FALSE (default): Close the brake of the axis.
  /// See Table 6-676 for bit assignment.
  ExternalAxesBrakeRelease : ExternalAxesFlags;
END_STRUCT
END_TYPE

// Library/POUs/Additional/MC_OpenBrake/Structures/OpenBrakeRecvData
{attribute 'pack_mode' := '1'} 
// ------------------------------------------------------------------------- 
//  SRCI Robot Library                                                
// ------------------------------------------------------------------------- 
//                                                                           
//  Object:      BrakeTestRecvData                                       
//  Author:      Thorsten Brach                                                
//  Date:        2024-06-01
//
//  Description:                                              
//   
//                                                                           
//  Copyright: 
//    (C) 2024 Thorsten Brach. All rights reserved                                                                                                                                            
//             Licensed under the LGPL-3.0 license.
//                                                                           
//  Disclaimer:                                                                           
//    This project is provided without any guarantee and can be used for   
//    private and commercial purposes. Any use is at the user’s 
//    own risk and responsibility.
//
// -------------------------------------------------------------------------
TYPE OpenBrakeRecvData EXTENDS RspHeader :
STRUCT
  /// TRUE when "OpenBrake" is active.
  Enabled                   : BYTE;  
  /// Indicates the brake release status of the main robot axes.
  /// • TRUE: The brake of the axis is opened.
  /// • FALSE: The brake of the axis is closed.
  /// See Table 6-735 for bit assignment
  RobotAxesBrakeReleased    : BYTE;
  /// Indicates the brake release status of the external robot axes.
  /// • TRUE: The brake of the axis is opened.
  /// • FALSE: The brake of the axis is closed/not supported
  /// See Table 6-735 for bit assignment
  ExternalAxesBrakeReleased : BYTE;
END_STRUCT
END_TYPE

// Library/POUs/Additional/MC_OpenBrake/Structures/OpenBrakeSendData
{attribute 'pack_mode' := '1'}
// ------------------------------------------------------------------------- 
//  SRCI Robot Library                                                
// ------------------------------------------------------------------------- 
//                                                                           
//  Object:      BrakeTestSendData                                       
//  Author:      Thorsten Brach                                                
//  Date:        2024-06-01
//
//  Description:                                              
//   
//                                                                           
//  Copyright: 
//    (C) 2024 Thorsten Brach. All rights reserved                                                                                                                                            
//             Licensed under the LGPL-3.0 license.
//                                                                           
//  Disclaimer:                                                                           
//    This project is provided without any guarantee and can be used for   
//    private and commercial purposes. Any use is at the user’s 
//    own risk and responsibility.
//
// -------------------------------------------------------------------------
TYPE OpenBrakeSendData EXTENDS CmdHeader:   
STRUCT
  /// Defines which brake of the robot axes must be released.
  /// • TRUE: Open the brake of the axis.
  /// • FALSE (default): Close the brake of the axis.
  RobotAxesBrakeRelease    : BYTE;
  /// Defines which brake of the external robot axis must be released.
  /// • TRUE: Open the brake of the axis.
  /// • FALSE (default): Close the brake of the axis.
  /// See Table 6-676 for bit assignment.
  ExternalAxesBrakeRelease : BYTE;
END_STRUCT
END_TYPE

// Library/POUs/Additional/MC_PathAccuracyMode/Structures/PathAccuracyModeOutCmd
{attribute 'pack_mode' := '1'} 
// ------------------------------------------------------------------------- 
//  SRCI Robot Library                                                
// ------------------------------------------------------------------------- 
//                                                                           
//  Object:      PathAccuracyModeOutCmd                                       
//  Author:      Thorsten Brach                                                
//  Date:        2024-06-22
//
//  Description:                                              
//   
//                                                                           
//  Copyright: 
//    (C) 2024 Thorsten Brach. All rights reserved                                                                                                                                            
//             Licensed under the LGPL-3.0 license.
//                                                                           
//  Disclaimer:                                                                           
//    This project is provided without any guarantee and can be used for   
//    private and commercial purposes. Any use is at the user’s 
//    own risk and responsibility.
//
// -------------------------------------------------------------------------
TYPE PathAccuracyModeOutCmd :
STRUCT
END_STRUCT
END_TYPE

// Library/POUs/Additional/MC_PathAccuracyMode/Structures/PathAccuracyModeParCmd
{attribute 'pack_mode' := '1'} 
// ------------------------------------------------------------------------- 
//  SRCI Robot Library                                                
// ------------------------------------------------------------------------- 
//                                                                           
//  Object:      PathAccuracyModeParCmd                                       
//  Author:      Thorsten Brach                                                
//  Date:        2024-06-22
//
//  Description:                                              
//   
//                                                                           
//  Copyright: 
//    (C) 2024 Thorsten Brach. All rights reserved                                                                                                                                            
//             Licensed under the LGPL-3.0 license.
//                                                                           
//  Disclaimer:                                                                           
//    This project is provided without any guarantee and can be used for   
//    private and commercial purposes. Any use is at the user’s 
//    own risk and responsibility.
//
// -------------------------------------------------------------------------
TYPE PathAccuracyModeParCmd :
STRUCT
END_STRUCT
END_TYPE

// Library/POUs/Additional/MC_PathAccuracyMode/Structures/PathAccuracyModeRecvData
{attribute 'pack_mode' := '1'} 
// ------------------------------------------------------------------------- 
//  SRCI Robot Library                                                
// ------------------------------------------------------------------------- 
//                                                                           
//  Object:      PathAccuracyModeRecvData                                       
//  Author:      Thorsten Brach                                                
//  Date:        2024-06-22
//
//  Description:                                              
//   
//                                                                           
//  Copyright: 
//    (C) 2024 Thorsten Brach. All rights reserved                                                                                                                                            
//             Licensed under the LGPL-3.0 license.
//                                                                           
//  Disclaimer:                                                                           
//    This project is provided without any guarantee and can be used for   
//    private and commercial purposes. Any use is at the user’s 
//    own risk and responsibility.
//
// -------------------------------------------------------------------------
TYPE PathAccuracyModeRecvData EXTENDS RspHeader :
STRUCT
  /// TRUE while PathAccuracyMode is active
  Enabled : BOOL;
END_STRUCT
END_TYPE

// Library/POUs/Additional/MC_PathAccuracyMode/Structures/PathAccuracyModeSendData
{attribute 'pack_mode' := '1'}
// ------------------------------------------------------------------------- 
//  SRCI Robot Library                                                
// ------------------------------------------------------------------------- 
//                                                                           
//  Object:      PathAccuracyModeSendData                                       
//  Author:      Thorsten Brach                                                
//  Date:        2024-06-22
//
//  Description:                                              
//   
//                                                                           
//  Copyright: 
//    (C) 2024 Thorsten Brach. All rights reserved                                                                                                                                            
//             Licensed under the LGPL-3.0 license.
//                                                                           
//  Disclaimer:                                                                           
//    This project is provided without any guarantee and can be used for   
//    private and commercial purposes. Any use is at the user’s 
//    own risk and responsibility.
//
// -------------------------------------------------------------------------
TYPE PathAccuracyModeSendData EXTENDS CmdHeader: 
STRUCT
  /// Set TRUE to activate monitoring of work areas
  Enable             : BOOL;
END_STRUCT
END_TYPE

// Library/POUs/Additional/MC_ReadCallSubprogramCyclic/Structures/ReadCallSubprogramCyclicOutCmd
{attribute 'pack_mode' := '1'} 
// ------------------------------------------------------------------------- 
//  SRCI Robot Library                                                
// ------------------------------------------------------------------------- 
//                                                                           
//  Object:      UnitMeasurementOutCmd                                       
//  Author:      Thorsten Brach                                                
//  Date:        2024-08-11
//
//  Description:                                              
//   
//                                                                           
//  Copyright: 
//    (C) 2024 Thorsten Brach. All rights reserved                                                                                                                                            
//             Licensed under the LGPL-3.0 license.
//                                                                           
//  Disclaimer:                                                                           
//    This project is provided without any guarantee and can be used for   
//    private and commercial purposes. Any use is at the user’s 
//    own risk and responsibility.
//
// -------------------------------------------------------------------------
TYPE ReadCallSubprogramCyclicOutCmd :
STRUCT
  /// Cyclic input data of subprogram
  Data : ARRAY[0..25] OF BYTE;
END_STRUCT
END_TYPE

// Library/POUs/Additional/MC_ReadCallSubprogramCyclic/Structures/ReadCallSubprogramCyclicParCmd
{attribute 'pack_mode' := '1'} 
// ------------------------------------------------------------------------- 
//  SRCI Robot Library                                                
// ------------------------------------------------------------------------- 
//                                                                           
//  Object:      UnitMeasurementParCmd                                       
//  Author:      Thorsten Brach                                                
//  Date:        2024-08-11
//
//  Description:                                              
//   
//                                                                           
//  Copyright: 
//    (C) 2024 Thorsten Brach. All rights reserved                                                                                                                                            
//             Licensed under the LGPL-3.0 license.
//                                                                           
//  Disclaimer:                                                                           
//    This project is provided without any guarantee and can be used for   
//    private and commercial purposes. Any use is at the user’s 
//    own risk and responsibility.
//
// -------------------------------------------------------------------------
TYPE ReadCallSubprogramCyclicParCmd :
STRUCT
END_STRUCT
END_TYPE

// Library/POUs/Additional/MC_ShiftPosition/Structures/ShiftPositionOutCmd
{attribute 'pack_mode' := '1'} 
// ------------------------------------------------------------------------- 
//  SRCI Robot Library                                                
// ------------------------------------------------------------------------- 
//                                                                           
//  Object:      ShiftPositionOutCmd                                       
//  Author:      Thorsten Brach                                                
//  Date:        2024-06-22
//
//  Description:                                              
//   
//                                                                           
//  Copyright: 
//    (C) 2024 Thorsten Brach. All rights reserved                                                                                                                                            
//             Licensed under the LGPL-3.0 license.
//                                                                           
//  Disclaimer:                                                                           
//    This project is provided without any guarantee and can be used for   
//    private and commercial purposes. Any use is at the user’s 
//    own risk and responsibility.
//
// -------------------------------------------------------------------------
TYPE ShiftPositionOutCmd :
STRUCT
  /// Tool index
  TransformedPosition       : RobotCartesianPosition;  
END_STRUCT
END_TYPE

// Library/POUs/Additional/MC_ShiftPosition/Structures/ShiftPositionParCmd
{attribute 'pack_mode' := '1'} 
// ------------------------------------------------------------------------- 
//  SRCI Robot Library                                                
// ------------------------------------------------------------------------- 
//                                                                           
//  Object:      ShiftPositionParCmd                                       
//  Author:      Thorsten Brach                                                
//  Date:        2024-06-22
//
//  Description:                                              
//   
//                                                                           
//  Copyright: 
//    (C) 2024 Thorsten Brach. All rights reserved                                                                                                                                            
//             Licensed under the LGPL-3.0 license.
//                                                                           
//  Disclaimer:                                                                           
//    This project is provided without any guarantee and can be used for   
//    private and commercial purposes. Any use is at the user’s 
//    own risk and responsibility.
//
// -------------------------------------------------------------------------
TYPE ShiftPositionParCmd :
STRUCT
  /// Define which method should be used to transform the position:
  Mode                      : TransformMode;
  /// Absolute coordinates of the position that will be transformed in the selected coordinate systems (see input parameter CoordinateSystem).
  Position                  : RobotCartesianPosition;
  /// Defines the reference frame ID to which the "Position" that will be transformed is relative.
  /// • 0: WCS (default)
  /// • 1..254: User frames
  FrameNo                   : USINT;
  /// Defines the reference frame ID to which the "TransformedPosition" should be relative.
  /// • 0: WCS (default)
  /// • 1..254: User frames
  TargetFrameNo             : USINT;
  /// Defines the frame data relevant for the transformation of the "Position". Relates to all "Mode" settings. 
  /// The parameter includes the Frame ID to which the origin of the shifting and rotation is relative and the cartesian position of the origin
  TransformationParameter_1 : FrameData;
  /// Relates to all "Mode" settings. Defines the enabled axis or plane as reference straight line or reference plain for the transformation
  TransformationParameter_2 : ReferenceElement;
  /// Defines the angle of rotation around the defined straight line. 
  /// Related to "Mode" with the setting "Rotate around Straight Line".
  RotationAngle             : REAL;  
END_STRUCT
END_TYPE

// Library/POUs/Additional/MC_ShiftPosition/Structures/ShiftPositionRecvData
{attribute 'pack_mode' := '1'} 
// ------------------------------------------------------------------------- 
//  SRCI Robot Library                                                
// ------------------------------------------------------------------------- 
//                                                                           
//  Object:      ShiftPositionRecvData                                       
//  Author:      Thorsten Brach                                                
//  Date:        2024-06-22
//
//  Description:                                              
//   
//                                                                           
//  Copyright: 
//    (C) 2024 Thorsten Brach. All rights reserved                                                                                                                                            
//             Licensed under the LGPL-3.0 license.
//                                                                           
//  Disclaimer:                                                                           
//    This project is provided without any guarantee and can be used for   
//    private and commercial purposes. Any use is at the user’s 
//    own risk and responsibility.
//
// -------------------------------------------------------------------------
TYPE ShiftPositionRecvData EXTENDS RspHeader :
STRUCT
  /// Tool index
  TransformedPosition : RobotCartesianPosition;  
END_STRUCT
END_TYPE

// Library/POUs/Additional/MC_ShiftPosition/Structures/ShiftPositionSendData
{attribute 'pack_mode' := '1'}
// ------------------------------------------------------------------------- 
//  SRCI Robot Library                                                
// ------------------------------------------------------------------------- 
//                                                                           
//  Object:      ShiftPositionSendData                                       
//  Author:      Thorsten Brach                                                
//  Date:        2024-06-22
//
//  Description:                                              
//   
//                                                                           
//  Copyright: 
//    (C) 2024 Thorsten Brach. All rights reserved                                                                                                                                            
//             Licensed under the LGPL-3.0 license.
//                                                                           
//  Disclaimer:                                                                           
//    This project is provided without any guarantee and can be used for   
//    private and commercial purposes. Any use is at the user’s 
//    own risk and responsibility.
//
// -------------------------------------------------------------------------
TYPE ShiftPositionSendData EXTENDS CmdHeader: 
STRUCT
  /// Defines the frame data relevant for the transformation of the "Position". Relates to all "Mode" settings. 
  /// The parameter includes the Frame ID to which the origin of the shifting and rotation is relative and the cartesian position of the origin
  TransformationParameter_1 : FrameData;
  /// Relates to all "Mode" settings. Defines the enabled axis or plane as reference straight line or reference plain for the transformation
  TransformationParameter_2 : ReferenceElement;
  /// Defines the angle of rotation around the defined straight line. 
  /// Related to "Mode" with the setting "Rotate around Straight Line".
  RotationAngle             : REAL;
  /// Define which method should be used to transform the position:
  Mode                      : TransformMode;
  /// Defines the reference frame ID to which the "Position" that will be transformed is relative.
  /// • 0: WCS (default)
  /// • 1..254: User frames
  FrameNo                   : USINT;
  /// Defines the reference frame ID to which the "TransformedPosition" should be relative.
  /// • 0: WCS (default)
  /// • 1..254: User frames
  TargetFrameNo             : USINT;
  /// Absolute coordinates of the position that will be transformed in the selected coordinate systems (see input parameter CoordinateSystem).
  Position                  : RobotCartesianPosition;
END_STRUCT
END_TYPE

